{attribute 'qualified_only'}
{attribute 'strict'}
TYPE E_General_ProcessCycle :
(
	
IDLE							,
CLOSE_PROCESS_DOOR				,
WAIT_CLOSE_PROCESS_DOOR			,
OPEN_PROCESS_DOOR				,
WAIT_OPEN_PROCESS_DOOR			,
EXTEND_PROCESS_CYLINDER			,
WAIT_EXTEND_PROCESS_CYLINDER	,
RETRACT_PROCESS_CYLINDER		,
WAIT_RETRACT_PROCESS_CYLINDER	,
HOLD_PART						,
WAIT_HOLD_PART					,
RELEASE_PART					,
WAIT_RELEASE_PART				,
LEAK_TEST_HEIGHT_CHECK			,
WAIT_LEAK_TEST_HEIGHT_CHECK		,
CAMERA_CHECK_PART_PRESENT		,
WAIT_CAMERA_CHECK_PART_PRESENT	,
PART_PRESENT_CHECK				,
VACUUM_CYLINDER_EXTENSION		,
WAIT_VACUUM_CYLINDER_EXTENSION	,
VACUUM_CYLINDER_RETRACTION		,
WAIT_VACUUM_CYLINDER_RETRACTION	,
CHECK_SEPTUM_POSITION			,
WAIT_CHECK_SEPTUM_POSITION		,
WAIT_TO_SAVE_DATA				,
WAIT_RESULTS					,
RESULTS							,
SAVE_DATA						,
SAVE_DATA2						,
CSV_NEST1						,
CSV_NEST2						,
WAIT_REJECT_PART				,
REJECT_CHUTE_FULL				,
PUCK_DEFINITION					,
NEST_CLEARING					,

RESET_ALL_CMD						

);
END_TYPE

(* stored: Version 1.1.0.1, ProductVersion 3.1.4026.18
   DUT E_General_ProcessCycle: Id {efc1fb3f-e466-425d-af8e-a4df616b7389} *)
